// TIA Portal V19 export
VAR_GLOBAL   // PLC tag table "MTRDIR"
END_VAR
